// TIA Portal V20 export
TYPE "typeEnMeterBits"
TITLE = Energy Meter Bits / Energy meter bits
// Struktur Energy Meter Bits / Structure energy meter bits
// stored: Access Published
   STRUCT
      startAcyclic { ExternalVisible := 'False'} : Bool;   // startAcyclic
      startAuto { ExternalVisible := 'False'} : Bool;   // startAuto
      resetMinMaxData { ExternalVisible := 'False'} : Bool;   // resetMinMaxData
      resetEnergyMeter { ExternalVisible := 'False'} : Bool;   // resetEnergyMeter
   END_STRUCT;
END_TYPE
